FUNCTION_BLOCK getBreadFromSensors
VAR_INPUT
	breadColor: INT;
	breadWeightClass: STRING;
END_VAR
VAR_OUTPUT
	breadTypeImageID: INT;
	breadInfo: STRING;
END_VAR
VAR	
END_VAR

IF breadColor = 0 AND breadWeightClass = 'medium' THEN
    breadTypeImageID := 1; // Toast
    breadInfo := 'White Toast';
ELSIF breadColor = 0 AND breadWeightClass = 'heavy' THEN
    breadTypeImageID := 2; // Baguette
    breadInfo := 'White Baguette';
ELSIF breadColor = 1 AND breadWeightClass = 'medium' THEN
    breadTypeImageID := 3; // Rye
    breadInfo := 'Dark Rye';
ELSIF breadColor = 1 AND breadWeightClass = 'light' THEN
    breadTypeImageID := 4; // Bagel
    breadInfo := 'Dark Bagel';
ELSE
    breadTypeImageID := 0;
    breadInfo := 'Unknown';
END_IF;

END_FUNCTION_BLOCK

(* stored: Version 1.1.0.1, ProductVersion 3.1.4024.15
   POU getBreadFromSensors: Id {b0184326-85ae-4124-afa8-224bf3630ad1}, SpecialFunc None *)
